// TIA Portal V17 export
// export: Created 2023-02-14T02:49:16.1277971Z, ExportSetting WithDefaults, DisplayName Totally Integrated Automation Portal, DisplayVersion V17, DisplayName TIA Portal Openness, DisplayVersion V17, DisplayName TIA Portal Teamcenter Gateway, DisplayVersion V17, DisplayName TIA Portal Version Control Interface, DisplayVersion V17, DisplayName SINAMICS Startdrive Advanced, DisplayVersion V17, DisplayName SINAMICS Startdrive G130, G150, S120, S150, SINAMICS MV, S210, DisplayVersion V17, DisplayName SINAMICS Startdrive G110M, G120, G120C, G120D, G120P, G115D, DisplayVersion V17, DisplayName STEP 7 Professional, DisplayVersion V17, DisplayName STEP 7 Safety, DisplayVersion V17, DisplayName WinCC Professional, DisplayVersion V17
DATA_BLOCK "THE2_From_Mixing_To_BT"   // DB199
{ S7_Optimized_Access := 'FALSE' }
VERSION : 0.1
// stored: AutoNumber false, DBAccessibleFromOPCUA true, DBAccessibleFromWebserver true, IsOnlyStoredInLoadMemory false, IsWriteProtectedInAS false
   VAR RETAIN
      HeartBeat : Bool;
      CIPRequest : Bool;
      MixProofFlip : Bool;
      Drain_valve : Bool;
      _free_4 : Bool;
      _free_5 : Bool;
      _free_6 : Bool;
      _free_7 : Bool;
      ProductAvailable : Bool;
      ProductTransferInProgress : Bool;
      _free_10 : Bool;
      _free_11 : Bool;
      _free_12 : Bool;
      _free_13 : Bool;
      _free_14 : Bool;
      _free_15 : Bool;
      _free_real2 : Real := 52.25618;
      _free_real6 : Real := 93.70135;
      _free_real10 : Real := 95.52147;
      _free_real14 : Real := 90.2006;
      _free_real18 : Real;
      _free_real22 : Real;
      _free_real26 : Real;
      _free_real30 : Real;
      ForTHE2_Byte1 : Byte;
      ForTHE2_Byte2 : Byte;
      ForTHE2_Byte3 : Byte;
      ForTHE2_Byte4 : Byte;
   END_VAR
BEGIN
END_DATA_BLOCK
